FUNCTION_BLOCK FB_MotionAxisCommonNC IMPLEMENTS I_MotionAxisCommon
VAR_INPUT
END_VAR
VAR_OUTPUT
END_VAR
VAR
    AxisRef : REFERENCE TO AXIS_REF;
    iPersistentDataStorage : I_PersistentDataStorage;
    iMotionLogger : I_MotionLogger;
    bCommandedMoveAbsolute : BOOL;
    // trying not to duplicate this vars in each derivation
    bCommandedMoveHome : BOOL;
    bInterrupted : BOOL;
    bHomeBusy: BOOL;
    bHomeDone : BOOL;
    bHomeInterrupted	: BOOL;
    bHomeError 			: BOOL;
    fHomePosition : LREAL :=0.0;
    fHomingSpeedsFast : LREAL;
    fHomingSpeedsSlow : LREAL;
    fHomingAcceleration : LREAL;
    fHomeOffset : LREAL;
    nHomeErrorID 		: UDINT;
    eHomingMethod : E_DS402HomingMethod;
END_VAR

{warning 'Add property implementation'}
PROPERTY AbortDone : BOOL
GET
END_GET
END_PROPERTY

{warning 'Add property implementation'}
PROPERTY AxisState : MC_AxisStates
GET
END_GET
END_PROPERTY

{warning 'Add method implementation '}
METHOD BacklashCompensation
VAR_INPUT
    User_Enable	: BOOL;
    Backlash	: LREAL;
    BakclashRampRatio	: LREAL := 10.0;
    DisableMode	: E_DISABLEMODE := E_DISABLEMODE.DisableModeHold;
END_VAR
END_METHOD

{warning 'Add property implementation'}
PROPERTY BufferMode : MC_BufferMode
SET
END_SET
END_PROPERTY

{warning 'Add property implementation'}
PROPERTY Busy : BOOL
GET
END_GET
END_PROPERTY

{warning 'Add property implementation'}
PROPERTY CommandAborted : BOOL
GET
END_GET
END_PROPERTY

{warning 'Add property implementation'}
PROPERTY CommandedHalt : BOOL
GET
END_GET
SET
END_SET
END_PROPERTY

{warning 'Add property implementation'}
PROPERTY CommandedMoveAbsolute : BOOL
GET
END_GET
SET
END_SET
END_PROPERTY

{warning 'Add property implementation'}
PROPERTY CommandedMoveHome : BOOL
GET
END_GET
SET
END_SET
END_PROPERTY

{warning 'Add property implementation'}
PROPERTY CommandedReset : BOOL
GET
END_GET
SET
END_SET
END_PROPERTY

{warning 'Add property implementation'}
PROPERTY EncoderCount : UDINT
GET
END_GET
END_PROPERTY

{warning 'Add property implementation'}
PROPERTY Error : BOOL
GET
END_GET
END_PROPERTY

{warning 'Add property implementation'}
PROPERTY ErrorID : UDINT
GET
END_GET
END_PROPERTY

{warning 'Add property implementation'}
PROPERTY ErrorMessage : STRING
GET
END_GET
END_PROPERTY

//FB_Init is always available implicitly and it is used primarily for initialization.
//The return value is not evaluated. For a specific influence, you can also declare the
//methods explicitly and provide additional code there with the standard initialization
//code. You can evaluate the return value.
METHOD FB_Init: BOOL
VAR_INPUT
    bInitRetains: BOOL; // TRUE: the retain variables are initialized (reset warm / reset cold)
    bInCopyCode: BOOL;  // TRUE: the instance will be copied to the copy code afterward (online change)

    AxisRef : REFERENCE TO AXIS_REF;
    iPersistentDataStorage : I_PersistentDataStorage;
    iMotionLogger : I_MotionLogger;
END_VAR
THIS^.AxisRef REF= AxisRef;
THIS^.iPersistentDataStorage := iPersistentDataStorage;
THIS^.iMotionLogger := iMotionLogger;
END_METHOD

{warning 'Add method implementation '}
METHOD Halt
VAR_INPUT
    Execute	: BOOL;
    Deceleration	: LREAL := 0.0;
    Jerk	: LREAL := 0.0;
    BufferMode	: MC_BufferMode := MC_BufferMode.MC_Aborting;
END_VAR
END_METHOD

{warning 'Add property implementation'}
PROPERTY HaltBufferMode : MC_BufferMode
GET
END_GET
SET
END_SET
END_PROPERTY

{warning 'Add property implementation'}
PROPERTY HaltBusy : BOOL
GET
END_GET
END_PROPERTY

{warning 'Add property implementation'}
PROPERTY HaltDeceleration : LREAL
GET
END_GET
SET
END_SET
END_PROPERTY

{warning 'Add property implementation'}
PROPERTY HaltDone : BOOL
GET
END_GET
END_PROPERTY

{warning 'Add property implementation'}
PROPERTY HaltErrorID : UDINT
GET
END_GET
END_PROPERTY

{warning 'Add property implementation'}
PROPERTY HaltJerk : LREAL
GET
END_GET
SET
END_SET
END_PROPERTY

{warning 'Add method implementation '}
METHOD Home
END_METHOD

{warning 'Add property implementation'}
PROPERTY HomeBusy : BOOL
GET
END_GET
END_PROPERTY

{warning 'Add property implementation'}
PROPERTY HomeDone : BOOL
GET
END_GET
END_PROPERTY

{warning 'Add property implementation'}
PROPERTY HomeError : BOOL
GET
END_GET
END_PROPERTY

{warning 'Add property implementation'}
PROPERTY HomeErrorID : UDINT
GET
END_GET
END_PROPERTY

{warning 'Add property implementation'}
PROPERTY HomeInterrupted : BOOL
GET
END_GET
END_PROPERTY

{warning 'Add property implementation'}
PROPERTY HomeMode : E_EpicsHomeCmd
GET
END_GET
SET
END_SET
END_PROPERTY

{warning 'Add property implementation'}
PROPERTY HomePosition : LREAL
GET
END_GET
SET
END_SET
END_PROPERTY

{warning 'Add property implementation'}
PROPERTY HomingMethod : E_DS402HomingMethod
GET
END_GET
SET
END_SET
END_PROPERTY

{warning 'Add property implementation'}
PROPERTY InTargetPosition : BOOL
GET
END_GET
END_PROPERTY

{warning 'Add property implementation'}
PROPERTY MeasuredAcceleration : LREAL
GET
END_GET
END_PROPERTY

{warning 'Add property implementation'}
PROPERTY MeasuredPosition : LREAL
GET
END_GET
END_PROPERTY

{warning 'Add property implementation'}
PROPERTY MeasuredPositionDiff : LREAL
GET
END_GET
END_PROPERTY

{warning 'Add property implementation'}
PROPERTY MeasuredVelocity : LREAL
GET
END_GET
END_PROPERTY

{warning 'Add property implementation'}
PROPERTY ModeOfOperation : SINT
GET
END_GET
SET
END_SET
END_PROPERTY

{warning 'Add method implementation '}
METHOD MoveAbsolute
VAR_INPUT
    Execute	: BOOL;
    Position	: LREAL;
    Velocity	: LREAL;
    Acceleration	: LREAL := 0.0;
    Deceleration	: LREAL := 0.0;
    Jerk	: LREAL := 0.0;
    BufferMode	: MC_BufferMode := MC_BufferMode.MC_Aborting;
END_VAR
END_METHOD

{warning 'Add property implementation'}
PROPERTY MoveAbsoluteBusy : BOOL
GET
END_GET
END_PROPERTY

{warning 'Add property implementation'}
PROPERTY MoveAbsoluteDone : BOOL
GET
END_GET
END_PROPERTY

{warning 'Add property implementation'}
PROPERTY MoveAbsoluteError : BOOL
GET
END_GET
END_PROPERTY

{warning 'Add property implementation'}
PROPERTY MoveAbsoluteErrorID : UDINT
GET
END_GET
END_PROPERTY

{warning 'Add property implementation'}
PROPERTY MoveAbsoluteTargetAcceleration : LREAL
GET
END_GET
SET
END_SET
END_PROPERTY

{warning 'Add property implementation'}
PROPERTY MoveAbsoluteTargetDeceleration : LREAL
GET
END_GET
SET
END_SET
END_PROPERTY

{warning 'Add property implementation'}
PROPERTY MoveAbsoluteTargetJerk : LREAL
GET
END_GET
SET
END_SET
END_PROPERTY

{warning 'Add property implementation'}
PROPERTY MoveAbsoluteTargetPosition : LREAL
GET
END_GET
SET
END_SET
END_PROPERTY

{warning 'Add property implementation'}
PROPERTY MoveAbsoluteTargetVelocity : LREAL
GET
END_GET
SET
END_SET
END_PROPERTY

{warning 'Add property implementation'}
PROPERTY MoveDone : BOOL
GET
END_GET
END_PROPERTY

{warning 'Add property implementation'}
PROPERTY MoveMode : E_EpicsMotorCmd
GET
END_GET
END_PROPERTY

{warning 'Add property implementation'}
PROPERTY Name : STRING
GET
END_GET
SET
END_SET
END_PROPERTY

{warning 'Add property implementation'}
PROPERTY NCParamsReadInit : BOOL
GET
END_GET
END_PROPERTY

{warning 'Add property implementation'}
PROPERTY NegativeMotionIsEnabled : BOOL
GET
END_GET
END_PROPERTY

{warning 'Add property implementation'}
PROPERTY PositiveMotionIsEnabled : BOOL
GET
END_GET
END_PROPERTY

{warning 'Add method implementation '}
METHOD Power
VAR_INPUT
    Enable	: BOOL;
    Enable_Positive	: BOOL;
    Enable_Negative	: BOOL;
    (* in percent from 0 to 100 *)
    Override	: LREAL := 100.0;
    BufferMode	: MC_BufferMode := MC_BufferMode.MC_Aborting;
END_VAR
END_METHOD

{warning 'Add property implementation'}
PROPERTY PowerEnable : BOOL
GET
END_GET
SET
END_SET
END_PROPERTY

{warning 'Add property implementation'}
PROPERTY PowerEnableNegative : BOOL
GET
END_GET
SET
END_SET
END_PROPERTY

{warning 'Add property implementation'}
PROPERTY PowerEnablePositive : BOOL
GET
END_GET
SET
END_SET
END_PROPERTY

{warning 'Add property implementation'}
PROPERTY PowerError : BOOL
GET
END_GET
END_PROPERTY

{warning 'Add property implementation'}
PROPERTY PowerErrorID : UDINT
GET
END_GET
END_PROPERTY

{warning 'Add property implementation'}
PROPERTY PowerIsEnabled : BOOL
GET
END_GET
END_PROPERTY

{warning 'Add property implementation'}
PROPERTY PowerOverride : LREAL
GET
END_GET
SET
END_SET
END_PROPERTY

{warning 'Add property implementation'}
PROPERTY PowerStatus : BOOL
GET
END_GET
END_PROPERTY

{warning 'Add property implementation'}
PROPERTY RefreshDelay : TIME
GET
END_GET
SET
END_SET
END_PROPERTY

{warning 'Add method implementation '}
METHOD Reset
END_METHOD

{warning 'Add property implementation'}
PROPERTY ResetBusy : BOOL
GET
END_GET
END_PROPERTY

{warning 'Add property implementation'}
PROPERTY ResetDone : BOOL
GET
END_GET
END_PROPERTY

{warning 'Add property implementation'}
PROPERTY ResetError : BOOL
GET
END_GET
END_PROPERTY

{warning 'Add property implementation'}
PROPERTY ResetErrorID : UDINT
GET
END_GET
END_PROPERTY

{warning 'Add property implementation'}
PROPERTY RestoreError : BOOL
GET
END_GET
END_PROPERTY

{warning 'Add property implementation'}
PROPERTY RestoreErrorID : UDINT
GET
END_GET
END_PROPERTY

{warning 'Add property implementation'}
PROPERTY SavedPosition : LREAL
GET
END_GET
END_PROPERTY

{warning 'Add property implementation'}
PROPERTY Servo : BOOL
GET
END_GET
SET
END_SET
END_PROPERTY

{warning 'Add method implementation '}
(*
    Check all post condition before updating bCommandedMoveAbsolute
    The implmentatation will depend on the axis type
    DS402 NC/Direct axis : Implementation need to check that the drive is in the correct mode before initaiting the move then set bCommandedMoveAbsolute
    MP NC axis : will immediately write to bCommandedMoveAbsolute
*)
METHOD StartMove : BOOL
VAR_INPUT
    MoveMode	: E_EpicsMotorCmd;
    CmdExecute	: BOOL;
END_VAR
END_METHOD

END_FUNCTION_BLOCK

(* stored: Version 1.1.0.1
   POU FB_MotionAxisCommonNC: Id {eafb0e6d-b2ea-4f78-9aba-c3a29595f5d4}, SpecialFunc None
   Property AbortDone: Id {99337b3e-e122-4163-92be-c9628a0747e8}
   Get Get: Id {383a9784-219f-4e54-9559-0dd2de571b7d}
   Property AxisState: Id {00ab01f4-c909-4ad9-9e19-e9e0f9b5c576}
   Get Get: Id {b317383e-7afa-40c6-a98f-ac1e887f076d}
   Method BacklashCompensation: Id {0a0ca488-9f96-4c1f-9d3a-bbfa4ab99ac5}
   Property BufferMode: Id {778add8f-aa83-44d1-8db7-3684a062acc7}
   Set Set: Id {a1314b17-0ce4-4ebc-9e50-5a5c2aeea488}
   Property Busy: Id {3e04a133-d7cd-4682-9539-088d1493ca08}
   Get Get: Id {89c375b7-fbd4-4a37-8c49-ec3a5634cada}
   Property CommandAborted: Id {af20a5b7-c8d4-43f8-b95a-4b2b8df5392e}
   Get Get: Id {dbfc2b2f-ed18-4e1f-87d5-78d10622d531}
   Property CommandedHalt: Id {7532149e-2f86-4bb6-8cd8-0e159001c3ba}
   Get Get: Id {122d030d-7ae5-4b97-bbfb-54524ec49430}
   Set Set: Id {86b73093-f7ea-44cf-b8d3-55addce2a862}
   Property CommandedMoveAbsolute: Id {5d6b4394-4ee5-492a-bf3c-01cf151ce1b9}
   Get Get: Id {3e323aa8-8d00-4f1b-8c04-154db30e1808}
   Set Set: Id {ec63e466-09ff-48af-8fa1-c1e90d6a1b5f}
   Property CommandedMoveHome: Id {de0efd29-d5b5-47fa-a1be-eb600582d68b}
   Get Get: Id {5098abdc-fcc5-4eec-9eed-a5a25f43be41}
   Set Set: Id {96e93ef3-a218-4db3-a294-2142a88ea1f2}
   Property CommandedReset: Id {5b9e06aa-579b-4e16-8232-f79e745f2df7}
   Get Get: Id {430a07fe-720c-46d6-8a5b-3688e0f1e2c2}
   Set Set: Id {9b0d82da-0753-484e-8582-0216b8df3f0d}
   Property EncoderCount: Id {eabc27cb-c902-40a5-bfe4-aed5042e2a84}
   Get Get: Id {542ffb94-245d-42c1-9b52-94c18cf97ec1}
   Property Error: Id {6ae4f138-4505-4260-99b9-f2596ca64ac5}
   Get Get: Id {c6fa7c5e-3579-48ca-8da6-d0146b325dbb}
   Property ErrorID: Id {27a094af-618b-4867-acb2-f7ffb313bd0b}
   Get Get: Id {1a4bbc2a-e119-458b-bcb8-2ee81013a018}
   Property ErrorMessage: Id {9af5a2bc-a4e8-4266-bb15-4baa0e5bad54}
   Get Get: Id {5ad44cdb-162a-4264-971f-44e290e47ac7}
   Method FB_Init: Id {e360ca1f-dc31-4e69-81cc-e5dafd90c4e3}
   Method Halt: Id {f9cd2505-bf39-4cdb-bfd3-2ffb8315325b}
   Property HaltBufferMode: Id {9848f165-e7b6-46a1-864d-7d06dd19a4c1}
   Get Get: Id {df29ea59-c561-4aa7-a2ee-b9f9c935f662}
   Set Set: Id {e0740993-1556-4730-8761-4b80162c1a0c}
   Property HaltBusy: Id {f67c3493-4c48-414f-97a1-c09a096755c5}
   Get Get: Id {bb29b96b-1330-46a1-b82b-3e9b8bd2aa09}
   Property HaltDeceleration: Id {a6f3fcc9-15dc-4238-bfaf-49cccc4599f7}
   Get Get: Id {6490be0d-879b-4238-92c8-d342bfded09f}
   Set Set: Id {5b63b882-38a0-4ce8-b61e-b0e9b389facc}
   Property HaltDone: Id {bbbad2d2-fd8a-4213-adc1-d9c0bd38f0c7}
   Get Get: Id {7ada0197-db3e-43e5-9a21-fb7c076b2bed}
   Property HaltErrorID: Id {f2a1da38-1c25-49e2-acbc-2f5bf529c6b0}
   Get Get: Id {d0c53c07-ccd3-4a73-bd56-958121fd4012}
   Property HaltJerk: Id {aa92d716-b371-4c64-9ba6-ce73ebf39cb5}
   Get Get: Id {309630a2-967c-432a-9375-54e3f2c8988c}
   Set Set: Id {cbaaf279-e540-4b66-b45b-87861b9bdcf4}
   Method Home: Id {cac9d768-0391-49f2-a7ee-360fa6f70aa3}
   Property HomeBusy: Id {8697f3d7-300a-4260-8339-0e1310a2412a}
   Get Get: Id {ba0e8a5f-95f3-40ab-8688-99e201c89c37}
   Property HomeDone: Id {e94ddfe1-664b-423b-bd2e-93398a4aa446}
   Get Get: Id {cd551903-d028-4eee-a169-692e0665c17d}
   Property HomeError: Id {2d495035-7eb7-47d1-a09a-eff3be362ac7}
   Get Get: Id {add61728-aef0-4738-ac99-8206c1d54e14}
   Property HomeErrorID: Id {84e05c19-5422-412e-a27f-651b5f4a77cc}
   Get Get: Id {745e273f-60f1-4219-b76e-41e70a096b87}
   Property HomeInterrupted: Id {5a08690d-0e09-44dd-a330-c6ea05cfdf43}
   Get Get: Id {e0b96cff-a419-47de-bcf7-158e9ff43abe}
   Property HomeMode: Id {68df4163-bf78-4f17-b574-d7bc076e6e3f}
   Get Get: Id {9e19e535-ae24-450f-8dcc-8ff6ccc2986f}
   Set Set: Id {63ac5308-27a5-4f31-b923-c1a67883aa33}
   Property HomePosition: Id {a97cb1eb-0848-4c6e-bc5c-b05e14afbbed}
   Get Get: Id {5a8f18da-65ae-40ae-a34b-884d9a3c2bf9}
   Set Set: Id {54f70e4a-4c37-46b1-b247-40dbef857ae6}
   Property HomingMethod: Id {4fe499b5-b8f2-45b7-b247-47c8d1ec4e23}
   Get Get: Id {b16845d3-e699-46ee-8fa7-23c81f10a142}
   Set Set: Id {97ca4597-9de7-42a7-a21a-874e20656b31}
   Property InTargetPosition: Id {700df9b8-1707-4308-abb5-d9ce6a8779b3}
   Get Get: Id {9761f3e9-b970-469b-866b-c551dab146e3}
   Property MeasuredAcceleration: Id {7ada6618-7c68-471e-af3b-2751ca321034}
   Get Get: Id {090a677a-f27d-4f6f-b42a-3dbcdf46b99d}
   Property MeasuredPosition: Id {9584aed0-4b87-4834-b9a0-22feefeeb692}
   Get Get: Id {7102c535-6f72-4319-9093-f57afa650018}
   Property MeasuredPositionDiff: Id {a53e7da6-2de7-4834-afbf-0ec4eb3c6637}
   Get Get: Id {b5893a80-7470-456b-bb29-6a7c42c36cff}
   Property MeasuredVelocity: Id {9fb897a1-44ed-47d2-b83a-1ca4eaa8903e}
   Get Get: Id {5501d9a4-ae37-40c3-8435-6dabab589307}
   Property ModeOfOperation: Id {342bf259-e743-4492-ad5c-153edb55ce1d}
   Get Get: Id {3de5762f-4682-429b-aea2-93bafb471ef0}
   Set Set: Id {768d0cab-0a88-45f4-9a6c-46dc63c985c8}
   Method MoveAbsolute: Id {0955f057-7eb6-41d7-8401-efa0950d5f47}
   Property MoveAbsoluteBusy: Id {e470117b-a320-4717-a34e-7b912b140d33}
   Get Get: Id {9b6e75db-c4c9-40cd-8811-cd3df50019fe}
   Property MoveAbsoluteDone: Id {7c6f6d1d-1c7e-418c-8cc6-b0d1b3a1a7f4}
   Get Get: Id {805af387-1171-4a10-8a57-d07f71451c1e}
   Property MoveAbsoluteError: Id {1a2759f4-77f3-4c86-a6aa-867d7c9c8373}
   Get Get: Id {0dcfabcc-6294-4aeb-bf40-11c8b7885835}
   Property MoveAbsoluteErrorID: Id {b6ea0536-dfef-432e-ab11-4f3ae0c8c9f4}
   Get Get: Id {1cd255b0-9003-47d5-829e-467c03b3d13b}
   Property MoveAbsoluteTargetAcceleration: Id {f46f61ad-9951-4f22-9156-919945390ceb}
   Get Get: Id {4f46d85d-8c2b-4464-864f-b7efc4d15f62}
   Set Set: Id {33af265b-60cd-40b0-bc93-473b5a8dd7ff}
   Property MoveAbsoluteTargetDeceleration: Id {edf505e7-f6d3-498d-8e64-a174131c0648}
   Get Get: Id {6b00674b-3764-4662-adfc-40ff716e820e}
   Set Set: Id {efd7bc12-80df-49ac-8923-3f0202cea5f7}
   Property MoveAbsoluteTargetJerk: Id {75a71f71-1831-45b9-a50e-3c7c552c0834}
   Get Get: Id {9908742b-3ac1-418a-b567-85de18029c70}
   Set Set: Id {364e9d4f-a284-40aa-a08f-ccbf2917bb30}
   Property MoveAbsoluteTargetPosition: Id {96022cd9-ac14-41d2-b5c2-0decf9a8b1e2}
   Get Get: Id {43260523-e96b-4420-8d3f-95517b8913b9}
   Set Set: Id {b44da972-111f-4083-a238-0f7ea17dc7b7}
   Property MoveAbsoluteTargetVelocity: Id {9ab1b669-e492-4b75-a292-59bbcc2229ae}
   Get Get: Id {e6ed8c0d-7008-440a-a9bd-756ae3dfd138}
   Set Set: Id {7dd38259-9483-47b4-9130-a3f8e603b1a3}
   Property MoveDone: Id {7217612a-991c-4a3d-925a-ec9638a6f1ff}
   Get Get: Id {79d9c879-8366-4a91-b1b1-b52cba679fb5}
   Property MoveMode: Id {ae7d75fc-2d1a-4a2e-bf73-5c86745d684c}
   Get Get: Id {e9ae0d07-c04d-45a9-8952-12845e2bd84c}
   Property Name: Id {4f28e4d5-8965-4aa8-a96e-6041117b81fa}
   Get Get: Id {08013349-5352-4f26-892f-12225a9b2754}
   Set Set: Id {81cdd04c-5036-4c88-8784-9a8031d25c53}
   Property NCParamsReadInit: Id {e4112f49-1416-4574-b622-3e07c96da7b9}
   Get Get: Id {33e00dea-f28e-4082-9bca-1e325cff2f7c}
   Property NegativeMotionIsEnabled: Id {5818072b-6397-4cef-a5c3-df26176e140e}
   Get Get: Id {cd68b34f-c7c2-4678-b63a-04f56463e7a4}
   Property PositiveMotionIsEnabled: Id {55f9e305-45c4-4a65-b57b-afd7a7dc0100}
   Get Get: Id {f3760e64-74fd-45ee-b106-b2698197d427}
   Method Power: Id {483b4736-b5f9-4b56-92da-d89e44e862d1}
   Property PowerEnable: Id {2bc3d398-4a95-4da7-9d57-b6232370eab4}
   Get Get: Id {f3ff8de3-91d8-41b6-97ac-0aea3db5a30a}
   Set Set: Id {1772e194-1ce0-475e-9fb1-d4f14a50fabf}
   Property PowerEnableNegative: Id {d6eeeddd-bdc9-40b2-84e0-3229c5f36627}
   Get Get: Id {f9e4dcb8-31c4-4f6f-8d69-eb9c39e8721f}
   Set Set: Id {bd29203f-c8f4-4fb7-8854-d455ed2776bc}
   Property PowerEnablePositive: Id {66702025-0418-4069-b9fc-b2ed114b4512}
   Get Get: Id {e77f59b4-07e3-4674-b10b-800f14f931ce}
   Set Set: Id {9a555c38-7965-4410-8c6e-f62fccd9ae41}
   Property PowerError: Id {aa8c297c-2ffd-45b4-9995-830c9acfae39}
   Get Get: Id {297d4b59-5584-4943-9ebd-5f5f1e104e54}
   Property PowerErrorID: Id {a03ea103-5c45-466e-8640-af86fbc76e75}
   Get Get: Id {c72de654-e963-49ab-ad38-654d99f28e1b}
   Property PowerIsEnabled: Id {bd3458b4-3a3c-4ac6-92e8-266de30b9183}
   Get Get: Id {4702760e-eb7b-4eac-a845-8ff8c1830e15}
   Property PowerOverride: Id {f231d4b3-cc65-49e2-9cd0-150a3d991114}
   Get Get: Id {62956b92-40cb-4263-b42c-20963af41481}
   Set Set: Id {d5d17e42-4cc9-499a-9ae2-876900f83e29}
   Property PowerStatus: Id {963a2400-9c66-4c17-9d1a-4eca775f9da4}
   Get Get: Id {1d963ddc-78cc-4324-b734-3ecb7c5d0c76}
   Property RefreshDelay: Id {376c85ec-acee-4ac4-8c69-9fc62f26cadf}
   Get Get: Id {75406b61-0ec5-40f4-8fb3-128efa9279f1}
   Set Set: Id {79b7f527-f347-4eb6-9ca9-b465746a49c9}
   Method Reset: Id {ab2b5a68-e6cd-47bc-aa3a-73d08162132e}
   Property ResetBusy: Id {08c3f7a4-9361-4547-b944-17d44319bad0}
   Get Get: Id {44bef986-18d1-46ac-88ad-14cca42013ee}
   Property ResetDone: Id {7ae4c7ba-2ba4-4cbd-b1f1-5b3dece2e38a}
   Get Get: Id {13b99075-a6ce-4445-81d8-e0e1dc3743d6}
   Property ResetError: Id {3d60f112-2328-43d2-b7fe-1418c30776d3}
   Get Get: Id {4b970aa1-6257-4e57-bd7b-5e4548f11afd}
   Property ResetErrorID: Id {b65200b8-dc2c-4003-83fb-60f2c53f80b1}
   Get Get: Id {3ebd7ff6-a118-4578-aaaf-27ace5cf2862}
   Property RestoreError: Id {fbd296dc-240f-4e9a-8e3e-7800239c94f3}
   Get Get: Id {eedb1e75-7411-4c78-af37-2a0aaa46aee0}
   Property RestoreErrorID: Id {152b9f7d-a790-462d-8d7f-025ed6ab877f}
   Get Get: Id {7d6a0e03-68de-4214-9452-43c7c6233cbd}
   Property SavedPosition: Id {4a68d335-2e33-48ce-a679-dc6e25767f56}
   Get Get: Id {b8b145ba-e5c6-4d8e-b132-cd1615e64e26}
   Property Servo: Id {282d0175-5a3f-4d8f-b961-2b3d9e6aff7b}
   Get Get: Id {288de6c0-7bae-40ba-94e5-611f7a8d9f1e}
   Set Set: Id {b7dfd3ed-89ed-465a-8575-a474be6e8503}
   Method StartMove: Id {273b2927-8144-4b20-a897-c504526ab82c} *)
